// TIA Portal V19 export
VAR_GLOBAL   // PLC tag table "Unit_DefaultTagTable_4"
END_VAR
